RoboDK station: Example_Camera.rdk

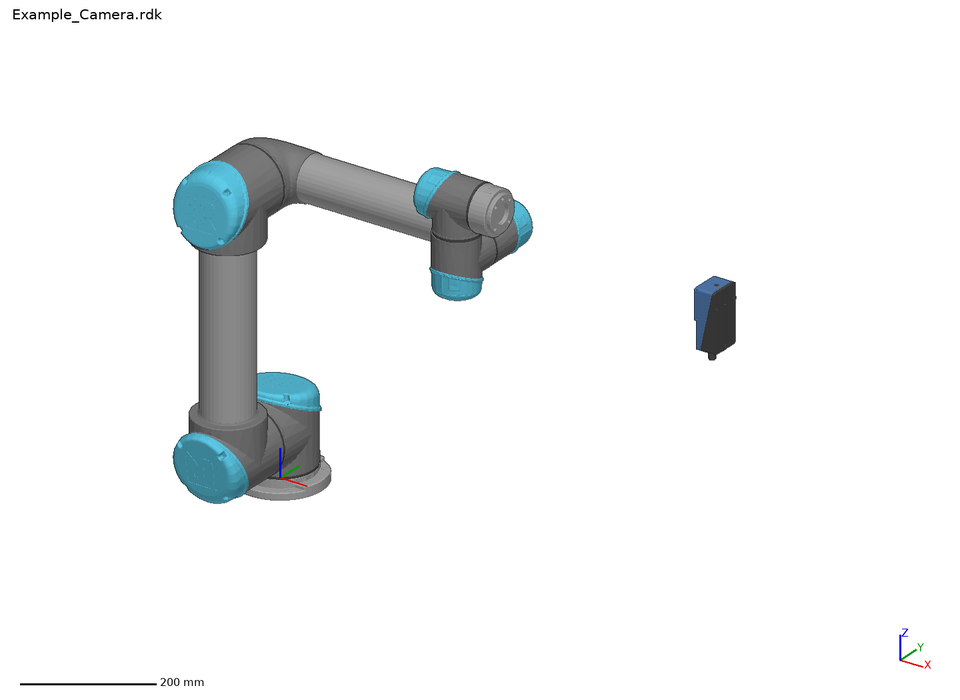
[picture v0: the station drawn from its stored meshes, robots at their saved joint values, targets as dots, program paths as lines]
Station Example_Camera (saved by RoboDK 5.3.5). Poses are relative to the parent item; angles as X-Y-Z fixed-axis rotations.
  - frame UR5 Base at (0, -229.88, -201.86) mm
    - robot UR5: 6 axes, payload 5 kg, reach 850 mm, repeatability 0.1 mm, weight 18.4 kg
        modified DH rows (alpha deg, a mm, theta deg, d mm): 0, 0, 0, 89.2; 90, 0, 180, 0; 0, 425, 0, 0; 0, 392.43, 0, 109; -90, 0, 0, 93.65; 90, 0, 180, 82
        joint limits [-360, -360, -360, -360, -360, -360] to [360, 360, 360, 360, 360, 360]; home [0, -90, -90, 0, 90, 0]; saved at [0, -90, -90, 0, 90, 0]
  - object SICK VSPP-5f2113 at (845.32, -351.76, 377.89) mm, rotated rx 0 ry -90 rz 0 deg, size 53 x 116 x 38 mm, geometry from Cam2D_SICK_VSPP_5F2113.sld
    - camera Camera1
  - Python program Prog1 (listed below)

--- Python program Prog1 ---
from robodk import robolink    # RoboDK API
from robodk import robomath    # Robot toolbox
RDK = robolink.Robolink()


cam_item = RDK.Item("Camera1")
if not cam_item.Valid():
    print('No camera..')
    quit()

snapshot_file='C:\FTPFiles\p1.jpg'
ret=RDK.Cam2D_Snapshot(snapshot_file,cam_item)
